FUNCTION_BLOCK C13336MppcWide EXTENDS C13336Mppc
VAR_INPUT
END_VAR
VAR_OUTPUT
END_VAR
VAR
	{attribute 'OPC.UA.DA' := '0'}
	_config : C13336MppcConfig;
	
	{attribute 'OPC.UA.DA' := '0'}
	_initDevice : BOOL;
	
	{attribute 'OPC.UA.DA.Access' := '0'}
    InputMppcWideStateSignal_1	AT %I* : BOOL;
	
	{attribute 'OPC.UA.DA.Access' := '0'}
    InputMppcWideStateSignal_2	AT %I* : BOOL;
	
	{attribute 'OPC.UA.DA' := '0'}
	_itemInit : INT;
	{attribute 'OPC.UA.DA' := '0'}
	_pulseGeneratorInit : TON;
	
	{attribute 'OPC.UA.DA' := '0'}
	_coeAccess : CoeAccess;
	{attribute 'OPC.UA.DA' := '0'}
	_initConfigSerialCom : BOOL;
	{attribute 'OPC.UA.DA' := '0'}
	_serialCom  : SerialCom(Prefix := Const.START_OF_TEXT, Suffix := Const.CARRIAGE_RETURN);
	{attribute 'OPC.UA.DA' := '0'}
	_refSerialCom : REFERENCE TO SerialCom(Prefix := Const.START_OF_TEXT, Suffix := Const.CARRIAGE_RETURN) := _serialCom;
		
END_VAR

IF NOT _raiseProperties THEN
	GetStateSignals();
END_IF

// Init device
SUPER^.InitDevice();

IF InitConfigSerialCom AND MppcActivate THEN
	THIS^.Status := TExecutionState.Ready;
ELSE
    THIS^.Status := TExecutionState.Error;	
END_IF

IF THIS^.Status = TExecutionState.Ready THEN
	SUPER^(Conf := _config, SerialCom := _serialCom, RefSerialCom := _refSerialCom);
END_IF

IF SUPER^._initDeviceBase THEN	
	IF NOT InitConfigSerialCom THEN
		ConfigureSerialCom();
	ELSIF THIS^.Status = TExecutionState.Ready THEN						
		_refSerialCom(TxBuffer:= HardwareGlobalVariables.TxBufferMppcWide, 
					  RxBuffer:= HardwareGlobalVariables.RxBufferMppcWide);		

		// Start Mppc to off 
		IF NOT _initDevice THEN
			InitDevice();
		END_IF					
	END_IF
END_IF

METHOD ConfigureSerialCom
VAR_INPUT
END_VAR

VAR
	Status: INT;
END_VAR
IF _coeAccess.CoeOperation.Ready THEN
	_logger.Information(_message.Reset().Append('Start configuration com serial').ToString());
END_IF;	

_coeAccess.CoeOperation.Start();
_coeAccess(SerialCommunication := _config.SerialCommunication);
	
IF _coeAccess.CoeOperation.Done THEN
	_coeAccess.SetDone();
	
	_Logger.Information(_message.Reset().
							Append('{').Append(TO_STRING(THIS^.Family)).Append('} : ').
							Append(' - Status : ').Append(TO_STRING(_coeAccess.Status)).ToString());
	InitConfigSerialCom := TRUE;
END_IF
 
IF _coeAccess.CoeOperation.Error THEN	
	_coeAccess.SetError(0);
	
	_Logger.Error(_message.Reset().
							Append('{').Append(TO_STRING(THIS^.Family)).Append('} : ').
							Append(' - Status : ').Append(TO_STRING(_coeAccess.Status)).ToString());
	InitConfigSerialCom := TRUE;
END_IF

THIS^.Status := _coeAccess.Status;
State := _coeAccess.Status;
END_METHOD

METHOD FB_init : BOOL
VAR_INPUT
	bInitRetains : BOOL; // if TRUE, the retain variables are initialized (warm start / cold start)
	bInCopyCode : BOOL;  // if TRUE, the instance afterwards gets moved into the copy code (online change)
	Config : C13336MppcConfig;
END_VAR
IF Config.IsEnabled THEN
	_config := Config;
	
	SUPER^._mppcConfig.Name := Config.Name;
	SUPER^._mppcConfig.DeviceID := Config.DeviceID;
	SUPER^._mppcConfig.IsEnabled := Config.IsEnabled;
	SUPER^._mppcConfig.LogLevel := Config.LogLevel;
	
	SUPER^.Name := Config.Name;
	SUPER^.DeviceID := Config.DeviceID;	
	THIS^.Family := DeviceFamily.MPPC;
		
	_Logger.Information(_message.Reset().Append('Init ').
							Append('{').Append(TO_STRING(THIS^.Family)).Append('} - ').
							Append('{').Append(TO_STRING(Config.Name)).Append('}').ToString());																													
END_IF
END_METHOD

METHOD GetStateSignals
VAR_INPUT
END_VAR
VAR
	{attribute 'OPC.UA.DA' := '0'}
	fibersCollector : STRING;
	{attribute 'OPC.UA.DA' := '0'}
	delimeter : STRING := ';';
	{attribute 'OPC.UA.DA' := '0'}
	stateSignal : STRING;	
	
END_VAR

fibersCollector := CONCAT(TO_STRING(EMppcCollector.WIDE), delimeter);

IF NOT InputMppcWideStateSignal_1 AND NOT InputMppcWideStateSignal_2 THEN
	stateSignal := CONCAT(fibersCollector, TO_STRING(EMppcStateModule.UNRECOVERABLE_ERROR));
ELSIF NOT InputMppcWideStateSignal_1 AND InputMppcWideStateSignal_2 THEN
	stateSignal := CONCAT(fibersCollector, TO_STRING(EMppcStateModule.AWAITING_COOLING_TEMP_STABLE));
ELSIF InputMppcWideStateSignal_1 AND NOT InputMppcWideStateSignal_2 THEN
	stateSignal := CONCAT(fibersCollector, TO_STRING(EMppcStateModule.AWAITING_HIGH_VOLTAGE_POWER_SUPPLY_STABLE));
ELSE
	stateSignal := CONCAT(fibersCollector, TO_STRING(EMppcStateModule.MODULE_OPERATING_NORMAL));
END_IF

IF stateSignal <> SUPER^.StateSignalsMsg THEN	
	SUPER^.StateSignalsMsg := stateSignal;
	SUPER^.GetStateSignals();
END_IF
END_METHOD

PROPERTY InitConfigSerialCom : BOOL
GET
InitConfigSerialCom := _initConfigSerialCom;
END_GET
SET
_initConfigSerialCom := InitConfigSerialCom;
END_SET
END_PROPERTY

METHOD InitDevice
VAR_INPUT
END_VAR
VAR	
END_VAR
IF NOT _initDevice THEN			
	IF _pulseGeneratorInit.Q THEN
		_pulseGeneratorInit(IN := FALSE, PT := T#10MS);
			
		CASE _itemInit OF
			0:  _logger.Information(_message.Reset().
								Append(_config.Name).
								Append(' - Start to on').ToString());		
				_itemInit := 1;
				
			1:  _outputVoltageOn := TRUE;			
				_initDevice := TRUE;
				_itemInit := 0;
		END_CASE
	ELSE
		_pulseGeneratorInit(IN := TRUE, PT := T#500MS);	
	END_IF
END_IF
END_METHOD

END_FUNCTION_BLOCK

(* stored: Version 1.1.0.1, ProductVersion 3.1.4024.12
   POU C13336MppcWide: Id {111a7122-6556-4c1a-aa0f-df797297d098}, SpecialFunc None
   Folder Commands: Id {bfc2ec1d-0b1f-426e-b808-03262d74be35}
   Method ConfigureSerialCom: Id {9adc588c-5e96-4382-8bbc-cd26a3f7e2a9}
   Method FB_init: Id {f74c4f58-0372-44ca-868c-74afb8e454fc}
   Method GetStateSignals: Id {21bd8d63-62e7-47dc-bc22-a35c5e68d48a}
   Property InitConfigSerialCom: Id {dda66ed7-bbc2-4c9f-bede-22f6907d2a8e}
   Get Get: Id {238b098a-aec8-4a3b-9a2f-ae612b6a1128}
   Set Set: Id {47cf8940-4731-447b-9ac1-1d9391219386}
   Method InitDevice: Id {c76989ba-65de-433a-9d4a-4875c40437d7} *)
